FUNCTION_BLOCK EL4021
VAR
	_io : EL4xx1_Data;
	{attribute addProperty Name "WcState"}
	_wcState : WcStateBase;
	{attribute addProperty Name "Info data"}
	_infoData : InfoDataAds;
END_VAR

PROPERTY IO : REFERENCE TO EL4xx1_Data
GET
IO REF= _io;
END_GET
END_PROPERTY

PROPERTY WcState : REFERENCE TO WcStateBase
GET
WcState REF= _wcState;
END_GET
END_PROPERTY

END_FUNCTION_BLOCK

(* stored: Version 1.1.0.1, ProductVersion 3.1.4024.9
   POU EL4021: Id {fd02f37b-5256-01ef-1e2a-39c08bbf731a}, SpecialFunc None
   Property IO: Id {3842a9bb-d6a2-0716-3d76-ad16a7243165}
   Get Get: Id {2f97d9bd-de49-0c77-05cc-7df6b5d49307}
   Property WcState: Id {3d74cd75-c694-0af9-0eb1-882023a84a3a}
   Get Get: Id {34b670d6-71cf-006b-0796-4596e9b60fea} *)
